# EPICS IOC start-up script: iocBoot/iocxxx/common.iocsh
### save_restore setup, change SAVE_PATH if you are having autosave manage its own NFS mount
iocshLoad("$(AUTOSAVE)/iocsh/autosave_settings.iocsh", "PREFIX=$(PREFIX), SAVE_PATH=$(TOP)/iocBoot/$(IOC), NUM_SEQ=12, SEQ_PERIOD=43200")
iocshLoad("$(AUTOSAVE)/iocsh/autosaveBuild.iocsh",     "PREFIX=$(PREFIX), BUILD_PATH=autosave")
iocshLoad("$(AUTOSAVE)/iocsh/save_restore.iocsh",      "PREFIX=$(PREFIX), POSITIONS_FILE=auto_positions, SETTINGS_FILE=auto_settings")

###
# specify directories in which to search for included request files
# Note that the vxWorks variables (e.g., 'startup') are from cdCommands
set_requestfile_path("$(ADCORE)/db")
set_requestfile_path("$(AUTOSAVE)/db")
set_requestfile_path("$(BUSY)/db")
set_requestfile_path("$(CALC)/db")
set_requestfile_path("$(CAMAC)/db")
set_requestfile_path("$(CAPUTRECORDER)/db")
set_requestfile_path("$(DAC128V)/db")
set_requestfile_path("$(DELAYGEN)/db")
set_requestfile_path("$(DXP)/db")
set_requestfile_path("$(DXPSITORO)/db")
set_requestfile_path("$(IP)/db")
set_requestfile_path("$(IP330)/db")
set_requestfile_path("$(IPUNIDIG)/db")
set_requestfile_path("$(LOVE)/db")
set_requestfile_path("$(LUA)/db")
set_requestfile_path("$(MCA)/db")
set_requestfile_path("$(MEASCOMP)/db")
set_requestfile_path("$(MODBUS)/db")
set_requestfile_path("$(MOTOR)/db")
set_requestfile_path("$(OPTICS)/db")
set_requestfile_path("$(QUADEM)/db")
set_requestfile_path("$(SSCAN)/db")
set_requestfile_path("$(SOFTGLUE)/db")
set_requestfile_path("$(SOFTGLUEZYNQ)/db")
set_requestfile_path("$(STD)/db")
set_requestfile_path("$(VAC)/db")
set_requestfile_path("$(VME)/db")
set_requestfile_path("$(YOKOGAWA_DAS)/db")
set_requestfile_path("$(TOP)/db")
set_requestfile_path("$(TOP)/xxxApp/Db")

# Debug-output level
save_restoreSet_Debug(0)

# devIocStats
dbLoadRecords("$(DEVIOCSTATS)/db/iocAdminSoft.db","IOC=$(PREFIX)")
# PV aliases change :: into :
# see https://github.com/epics-modules/xxx/issues/30
dbLoadRecords("$(TOP)/xxxApp/Db/iocAdminSoft_aliases.db","P=$(PREFIX)")

### Scan-support software
iocshLoad("$(SSCAN)/iocsh/sscan.iocsh", "PREFIX=$(PREFIX), MAX_PTS=1000, REQ_FILE=saveData.req")
iocshLoad("$(AUTOSAVE)/iocsh/configMenu.iocsh", "PREFIX=$(PREFIX),CONFIG=scan1")

### Stuff for user programming ###
iocshLoad("$(CALC)/iocsh/userCalc.iocsh", "PREFIX=$(PREFIX), ARRAY_SIZE=8000")

# Load 10 more of all the user calcs, N=1 creates usercalcs 10-19
iocshLoad("$(CALC)/iocsh/userCalc_extra.iocsh", "PREFIX=$(PREFIX), N=1, ARRAY_SIZE=8000")

# Load 20 userScripts
#dbLoadRecords("$(LUA)/luaApp/Db/luascripts10.db", "P=$(PREFIX), R=set1:")
#dbLoadRecords("$(LUA)/luaApp/Db/luascripts10.db", "P=$(PREFIX), R=set2:")

# string sequence (sseq) records
iocshLoad("$(CALC)/iocsh/sseq.iocsh", "PREFIX=$(PREFIX), INSTANCE=ES:")

# busy record
dbLoadRecords("$(BUSY)/busyApp/Db/busyRecord.db", "P=$(PREFIX),R=mybusy1")
dbLoadRecords("$(BUSY)/busyApp/Db/busyRecord.db", "P=$(PREFIX),R=mybusy2")

### Load database record for alive heartbeating support.
# IOCNM is name of IOC, RHOST specifies the remote server accepting hearbeats
dbLoadRecords("$(ALIVE)/aliveApp/Db/alive.db", "P=$(PREFIX),IOCNM=$(IOC),RHOST=164.54.100.11")
dbLoadRecords("$(ALIVE)/aliveApp/Db/aliveMSGCalc.db", "P=$(PREFIX)")

# Miscellaneous PV's, such as burtResult
dbLoadRecords("$(STD)/stdApp/Db/misc.db","P=$(PREFIX)")
